FUNCTION_BLOCK Digital_Input
VAR_INPUT
	Input		: BOOL;
END_VAR
VAR_OUTPUT
END_VAR
VAR
END_VAR

PROPERTY PUBLIC Status : BOOL
GET
Status := Input;
END_GET
END_PROPERTY

END_FUNCTION_BLOCK

(* stored: Version 1.1.0.1, ProductVersion 3.1.4024.10
   POU Digital_Input: Id {96ecf1fb-507a-4986-9a07-9744e0d850f9}, SpecialFunc None
   Property Status: Id {48516cb1-9761-485e-9dbb-8165f63de4be}
   Get Get: Id {b8c0b06c-26a8-4cb1-88a4-f6a471440adb} *)
